(* PLC project OOP_Curso, Beckhoff Automation GmbH TwinCAT PLC Control 3.5.13.21 *)
(* stored: creationDateTime 2023-02-07T16:35:16.3639657, modificationDateTime 2023-02-07T16:35:16.3717731 *)

FUNCTION_BLOCK Coche_3
VAR_INPUT
	bInput : BOOL;
END_VAR
VAR_OUTPUT
	bOutput : BOOL;
END_VAR
VAR_IN_OUT
	bInOut : BOOL;
END_VAR
VAR
	_Marca : STRING;
	_Color : STRING;
	accion : STRING;
END_VAR

            
          

METHOD PUBLIC Acelerar
                  accion := 'acelerar';
                
END_METHOD

METHOD PUBLIC Conducir
                  accion := 'conducir';
                
END_METHOD

METHOD PUBLIC Frenar
                  accion := 'frenar';
                
END_METHOD

METHOD FB_init : BOOL
VAR_INPUT
	bInitRetains : BOOL; // if TRUE, the retain variables are initialized (warm start / cold start)
	bInCopyCode : BOOL;  // if TRUE, the instance afterwards gets moved into the copy code (online change)
	Marca        : STRING;
	Color        : STRING;
END_VAR
                  THIS^._Marca := Marca;
THIS^._Color := Color;
                
END_METHOD

METHOD FB_reinit : BOOL
VAR_INPUT
END_VAR
                  
                
END_METHOD

METHOD FB_exit : BOOL
VAR_INPUT
	bInCopyCode : BOOL; // if TRUE, the exit method is called for exiting an instance that is copied afterwards (online change).
END_VAR
                  
                
END_METHOD

PROPERTY PUBLIC Color : STRING
GET
                    Color := _Color;
                  
END_GET
SET
                    _Color := Color;
                  
END_SET
END_PROPERTY

PROPERTY PUBLIC Marca : STRING
GET
                    Marca := _Marca;
                  
END_GET
SET
                    _Marca := Marca;
                  
END_SET
END_PROPERTY
END_FUNCTION_BLOCK

PROGRAM _03_Clase_y_Objetos
VAR
	// tenemos la Clase Coche y la instanciamos y obtenemos los Objetos: Mercedes, Bmw y Audi.
	Mercedes : Coche_3(Marca:= 'Mercedes', Color := 'Azul');
	
	Color : STRING;
	Marca : STRING;
	
	Acelerar : BOOL;
	Conducir:  BOOL;
	Frenar  : BOOL;
	
	CambiarColor : BOOL;
END_VAR

            //Objeto Mercedes
//llamadas a sus métodos.
IF Acelerar THEN
	Mercedes.Acelerar();
	Acelerar := FALSE;
END_IF

IF Conducir THEN
	Mercedes.Conducir();
	Conducir := FALSE;
END_IF

IF Frenar THEN
	Mercedes.Frenar();
	Frenar := FALSE;
END_IF

//llamadas a sus propiedades.
//Mercedes.Marca := 'Mercedes';
IF CambiarColor THEN
	Mercedes.Color := 'Negro';
	CambiarColor := FALSE;
END_IF

Color := Mercedes.Color;

          
END_PROGRAM
